ABB RobotStudio station: HandTracking_gripper_2.0.rspag

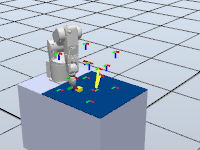
--- station ---
Station HandTrackingWithGripper (saved by RobotStudio 7.0.8743.626)
Controller Controller1, task T_ROB1: task frame (RAPID world) sits at (-300, 0, 800) mm in the station
Controller Controller1
  mechanical unit ROB_1: IRB1200_7_70_STD_02, 6 joints, base frame (0, 0, 0) mm
Layout (positions relative to the parent item):
  - IRB1200_7_70_STD_02 [mechanism, from Robots\IRB1200_7_70_STD_02.rslib] at (-300, 0, 800) mm; joint values [-0.4483, 0.9444, 0.5545, 0, 0.0719, 2.6932] (rad or m)
  - Stojalo3 [part] at (0, -390, 400) mm
  - Part_1 [part]
  - Smart_Gripper_Servo_Fingers_2_2 [mechanism] at (16, -152, 975.2) mm, rotated rx -180 ry 0 rz 0 deg; joint values [0.025] (rad or m)
      TCP Servo at (0, 0, 114.2) mm
      links: HandBase, DownFinger, UpFinger, VacuumOne, VacuumTwo
  - Part_2 [part] at (-100, 0, 0) mm
  - Part_3 [part] at (32.03, -118.48, 843.64) mm, rotated rx 0 ry 90 rz -90 deg
Attachment: Smart_Gripper_Servo_Fingers_2_2 is attached to IRB1200_7_70_STD_02 / Link6
EventTableEntry 1057: Group=, Trigger=DoFingers 1058, Actions=[EventTableActionMechanicalPose 1059], Comment=, ActivationMode=2, Cyclic=false
EventTableTriggerIO 1058: IOValue=[1], IRC5Controller=? -1, Operator=0, SignalSource=Controller1 515
EventTableActionMechanicalPose 1059: VirtualSignal=, Mechanism=Smart_Gripper_Servo_Fingers_2_2 1049, ToPoseName=Zaprto, VirtualSignalValue=[1]
EventTableEntry 1060: Group=, Trigger=DoFingers 1061, Actions=[EventTableActionMechanicalPose 1062], Comment=, ActivationMode=2, Cyclic=false
EventTableTriggerIO 1061: IOValue=[0], IRC5Controller=? -1, Operator=0, SignalSource=Controller1 515
EventTableActionMechanicalPose 1062: VirtualSignal=, Mechanism=Smart_Gripper_Servo_Fingers_2_2 1049, ToPoseName=Odprto, VirtualSignalValue=[1]
EventTableTriggerIO 1114: IOValue=[1], IRC5Controller=? -1, Operator=0, SignalSource=Controller1 515
EventTableTriggerIO 1115: IOValue=[0], IRC5Controller=? -1, Operator=0, SignalSource=Controller1 515
EventTableTriggerIO 1134: IOValue=[1], IRC5Controller=? -1, Operator=0, SignalSource=Controller1 515
EventTableTriggerIO 1135: IOValue=[0], IRC5Controller=? -1, Operator=0, SignalSource=Controller1 515
EventTableEntry 1193: Group=, Trigger=EventTableTriggerCustom 1194, Actions=[EventTableActionMove 1195], Comment=, ActivationMode=1, Cyclic=false
EventTableTriggerCustom 1194: Time=0, TriggerType=Timer
EventTableActionMove 1195: Object=Part_3 1203, GlobalTransform=[X=3.74915180455534E-33, Y=-6.12303176911189E-17, Z=-1, W=0, X=1, Y=6.12303176911189E-17, Z=0, W=0, X=6.12303176911189E-17, Y=-1, Z=6.12303176911189E-17, W=0, X=0.144379, Y=0, Z=0.86, W=1]
EventTableEntry 1196: Group=, Trigger=DoFingers 1197, Actions=[EventTableActionAttach 1198], Comment=, ActivationMode=2, Cyclic=false
EventTableTriggerIO 1197: IOValue=[1], IRC5Controller=? -1, Operator=0, SignalSource=Controller1 515
EventTableActionAttach 1198: AttachmentParent=Smart_Gripper_Servo_Fingers_2_2 1049, AttachmentChild=Part_3 1203, MountObject=false, Offset=[X=1, Y=0, Z=0, W=0, X=0, Y=1, Z=0, W=0, X=0, Y=0, Z=1, W=0, X=0, Y=0, Z=0, W=1], FlangeIndext=0, FindNearest=false
EventTableTriggerIO 1199: IOValue=[0], IRC5Controller=? -1, Operator=0, SignalSource=Controller1 515
EventTableEntry 1200: Group=, Trigger=DoFingers 1199, Actions=[EventTableActionDetach 1201], Comment=, ActivationMode=2, Cyclic=false
EventTableActionDetach 1201: AttachmentParent=Smart_Gripper_Servo_Fingers_2_2 1049, AttachmentChild=Part_3 1203
Targets, tools, work objects and paths stored in the station and not in the controller backup, written as RAPID:
! task T_ROB1
MODULE Module1
  CONST robtarget Target_30:=[[590,-205,410],[0,1,0,0],[-1,0,1,0],[9E+09,9E+09,9E+09,9E+09,9E+09,9E+09]];
  CONST robtarget Target_40:=[[590,195,410],[0,1,0,0],[0,0,-2,0],[9E+09,9E+09,9E+09,9E+09,9E+09,9E+09]];
  CONST robtarget Target_50:=[[190,195,410],[0,1,0,0],[0,0,0,0],[9E+09,9E+09,9E+09,9E+09,9E+09,9E+09]];
  CONST robtarget Target_60:=[[190,-205,10],[0,1,0,0],[0,0,0,0],[9E+09,9E+09,9E+09,9E+09,9E+09,9E+09]];
  CONST robtarget Target_70:=[[590,-205,10],[0,1,0,0],[0,0,0,0],[9E+09,9E+09,9E+09,9E+09,9E+09,9E+09]];
  CONST robtarget Target_80:=[[590,195,10],[0,1,0,0],[0,0,-2,0],[9E+09,9E+09,9E+09,9E+09,9E+09,9E+09]];
  CONST robtarget Target_90:=[[190,195,10],[0,1,0,0],[0,0,0,0],[9E+09,9E+09,9E+09,9E+09,9E+09,9E+09]];
  CONST robtarget Target_100:=[[108.00000974,170.999988771,-391.039697267],[0.000000118,0.000000013,0.70710678,0.707106782],[0,-1,2,0],[9E+09,9E+09,9E+09,9E+09,9E+09,9E+09]];
  CONST robtarget Target_110:=[[139.253700517,269.955882709,-327.170794361],[-0.000000081,0.000000036,0.707106783,0.707106779],[0,-1,-2,0],[9E+09,9E+09,9E+09,9E+09,9E+09,9E+09]];
ENDMODULE


--- Backups/Controller1/RAPID/TASK1/PROGMOD/Module1.mod ---
MODULE Module1
	PERS tooldata Servo:=[TRUE,[[0,0,114.2],[1,0,0,0]],[0.215,[8.7,12.3,49.2],[1,0,0,0],0.00021,0.00024,0.00009]];
	PERS wobjdata podlaga:=[FALSE,TRUE,"",[[590,-205,410],[0,0,-0.707106781,0.707106781]],[[0,0,0],[1,0,0,0]]];
    PERS num bReachable:=1;
    VAR num operatingmode:=1;
    VAR num waitpaint:=0;
    CONST robtarget home:=[[481.999971829,62.000001385,239.000022114],[-0.000000003,1,-0.000000021,0.000000068],[0,0,2,0],[9E+09,9E+09,9E+09,9E+09,9E+09,9E+09]];
    CONST robtarget Target_10:=[[490,-5,10],[0,0,1,0],[-1,0,-1,0],[9E+09,9E+09,9E+09,9E+09,9E+09,9E+09]];
    CONST robtarget Target_20:=[[205.90937827,223.382688175,387.01986369],[0.000000404,-0.00000012,0.707106786,0.707106776],[-1,-1,1,0],[9E+09,9E+09,9E+09,9E+09,9E+09,9E+09]];
    CONST robtarget TEsstarger:=[[181,225,-276],[0,0,0.707107,0.707107],[-1,-1,1,0],[9E+9,9E+9,9E+9,9E+9,9E+9,9E+9]];
    VAR num helpconfig:=0;
    VAR robtarget helprobottarget;
     VAR confdata cfgData;










     PROC main()
        VAR socketdev server_socket;
        VAR socketdev client_socket;
        VAR string receive_string;
        VAR string receive_string2;
        VAR string client_ip;
        VAR robtarget mytr;
        VAR string myIP:= "127.0.0.1"; !same as in config.py !!!





        SocketCreate server_socket;
        SocketBind server_socket,myIP, 55555;
        SocketListen server_socket;

        ConfL\Off;
        ConfJ\Off;
        SingArea \Wrist;

        MoveJ home,v1000,z30,Servo\WObj:=wobj0;


        ! Waiting for a connection request
         SocketAccept server_socket, client_socket\ClientAddress:=client_ip\Time:=WAIT_MAX;
         SocketSend client_socket \Str :="Robot at position "+TargetToString(home);

        WHILE TRUE DO
            !waiting to recive
            SocketReceive client_socket \Str := receive_string2;

            IF receive_string2="g" THEN
                !operating mode is in xy plane
               ! operatingmode:=0;

                IF DoFingers=0 THEN

                    SetDO DoFingers,1;
                     SocketSend client_socket \Str :="Robot grabbing";

                ELSEIF DoFingers=1 THEN
                    SetDO DoFingers,0;
                     SocketSend client_socket \Str :="Robot realising";


                ENDIF

                !TPWrite"moving set to XY plane now";


             ELSEIF receive_string2="xy" THEN
                !operating mode is in xy plane
                operatingmode:=0;
                SocketSend client_socket \Str :="operating in xy now";

                !TPWrite"moving set to XY plane now";

            ELSEIF receive_string2="xyz" THEN
                !operating mode is in xyz plane
                operatingmode:=1;
                waitpaint:=0;
                SocketSend client_socket \Str :="operating in xyz now";
                !TPWrite"moving set to XYZ now !";



            ELSE
                !MOVE

                 mytr:= StringToTargetFromxy(receive_string2); !get target from string
                 move mytr;!check if is reachable then move

            ENDIF


        ENDWHILE
        MoveJ home,v1000,z100,Servo\WObj:=wobj0;
        MoveL Target_10,v1000,z100,Servo\WObj:=wobj0;


    ERROR
        IF ERRNO=ERR_SOCK_TIMEOUT THEN
            RETRY;

        ELSEIF ERRNO=ERR_SOCK_CLOSED THEN

        SocketCreate server_socket;
        SocketBind server_socket, myIP, 55555;
        SocketListen server_socket;
            RETRY;
        ELSE
            RETRY;

        ENDIF
    UNDO
        SocketClose server_socket;
        SocketClose client_socket;
    ENDPROC


     FUNC robtarget create_robtarget(pos position)
       RETURN [position,[0,0,0.707106781,0.707106781],cfgData,[9E9,9E9,9E9,9E9,9E9,9E9]];
    ENDFUNC

    FUNC string TargetToString(robtarget target)
    VAR string tmpString;
    !pos data
    tmpString:=NumToStr (target.trans.x,0);
    AddToString tmpString,target.trans.y;
    AddToString tmpString, target.trans.z;
    ! orient data
    AddToString tmpString, target.rot.q1;
    AddToString tmpString, target.rot.q2;
    AddToString tmpString, target.rot.q3;
    AddToString tmpString, target.rot.q4;
    ! conf data
    AddToString tmpString, target.robconf.cf1;
    AddToString tmpString, target.robconf.cf4;
    AddToString tmpString, target.robconf.cf6;
    AddToString tmpString, target.robconf.cfx;
RETURN tmpString;
ENDFUNC

FUNC robtarget StringToTarget(string value)
    !CAN BE USED IF OREANTATIONS ARE NEEDED CURENTLY NOT USED
VAR robtarget tmpTarget;
VAR bool bResult;
VAR num posX;
VAR num posY;
VAR num posZ;
VAR num posQ1;
VAR num posQ2;
VAR num posQ3;
VAR num posQ4;
VAR num poscf1;
VAR num poscf4;
VAR num poscf6;
VAR num poscfx;
! Find split positions in string

posX:=StrFind (value, 1,";");
posY:=StrFind (value, posX+1,";");
posZ:=StrFind (value, posY+1,";");
posQ1:=StrFind (value, posZ+1,";");
posQ2:=StrFind(value, posQ1+1,";");
posQ3:=StrFind (value,posQ2+1,";");
posQ4:=Strfind(value, posQ3+1,";");
poscf1:=StrFind(value, posQ4+1,";");
poscf4:=StrFind(value, poscf1+1,";");
poscf6:=StrFind(value, poscf4+1,";");
poscfx:=StrFind(value,poscf6+1, ";");
! read all strings
! pos data
bResult:=StrToval(StrPart(value,1,posX-1), tmpTarget.trans.x);
bResult:=StrToVal(StrPart(value,posX+1, posY-posX-1), tmpTarget.trans.y);
bResult:=StrToVal(StrPart(value,posY+1, posZ-posY -1), tmpTarget.trans.z);
! orient data
bResult:=StrToVal(StrPart(value, posZ+1, posQ1-posz-1), tmpTarget.rot.q1);
bResult:=StrToval (StrPart(value,posQ1+1, posQ2-posQ1-1), tmpTarget.rot.q2);
bResult:=StrToVal(StrPart(value,posQ2+1, posQ3-posQ2-1), tmpTarget.rot.q3);
bResult:=StrToVal(StrPart(value,posQ3+1,posQ4-posQ3-1), tmpTarget.rot.q4);
! conf data
bResult:=StrToVal(StrPart(value,posQ4+1, poscf1-posQ4-1), tmpTarget.robconf.cf1);
bResult:=StrToVal(StrPart(value, poscf1+1,poscf4-poscf1-1), tmpTarget.robconf.cf4);
bResult:=StrToval(StrPart(value,poscf4+1,poscf6-poscf4-1), tmpTarget.robconf.cf6);
bResult:=StrToVal(StrPart(value,poscf6+1,poscfx-poscf6-1), tmpTarget.robconf.cfx);
RETURN tmpTarget;

ERROR
    !RETURN !Target_20;



ENDFUNC

FUNC robtarget StringToTargetFromxy(string value)
VAR pos tmpPos;
VAR robtarget tmpTarget;
VAR bool bResult;
VAR num posX;
VAR num posY;
VAR num posZ;
VAR num xxx;
VAR num yyy;
VAR num zzz:=-330;
! Find split positions in string

posX:=StrFind (value, 1,";");
posY:=StrFind (value, posX+1,";");
IF operatingmode=1 THEN
posZ:=StrFind (value, posY+1,";");
ENDIF

! pos data
bResult:=StrToval(StrPart(value,1,posX-1), tmpPos.x);

tmpPos.x:=tmpPos.x;

bResult:=StrToVal(StrPart(value,posX+1, posY-posX-1), tmpPos.y);

tmpPos.y:=tmpPos.y;

IF operatingmode=1 THEN
bResult:=StrToVal(StrPart(value,posY+1, posZ-posY -1), tmpPos.z);

tmpPos.z:=-tmpPos.z;

ELSE
tmpPos.z:=zzz; !z is set to 0
ENDIF
tmpTarget:=create_robtarget(tmpPos);
RETURN tmpTarget;

ERROR
   ! RETURN Target_20;!middle target of error
ENDFUNC

PROC AddToString(INOUT string inString,num value)
inString:=inString+";"+NumToStr(value,0);
ENDPROC

PROC move(robtarget target)
     VAR bool aotoconfiggg;
     VAR bool precheck:=FALSE;
     precheck:=simplecheck(target,Servo);

     !IF precheck=FALSE THEN
    !aotoconfiggg:= calcconfiguration(target,Servo);
     !IF aotoconfiggg=TRUE THEN
      !   target.robconf:=cfgData;

    !CheckReachable target,Servo;
     !      IF bReachable=2 THEN
                !notreachable
      !          TPWrite"not reachable";
       !    ELSEIF bReachable=1 THEN
                !reachable start moving
        !        MoveJ target,v2000,z10,Servo\WObj:=podlaga;

                !move target;
         ! ENDIF
          ! ELSE
        ! RETURN;
     !ENDIF

     !ELSE
          MoveJ target,v2000,z10,Servo\WObj:=podlaga;

     !ENDIF

    ERROR
        TPWrite"error in move";
        TRYNEXT;

ENDPROC


 PROC CheckReachable(robtarget myRobtarget,PERS tooldata ToolReach1,\PERS wobjdata WobjReach1)

      VAR jointtarget jntReach1;



      bReachable:=1;

            jntReach1:=CalcJointT(myRobtarget,ToolReach1);

      RETURN;
      ERROR


         IF ERRNO=ERR_OUTSIDE_REACH THEN

                bReachable:=2;
               TRYNEXT;

        ENDIF
         IF ERRNO=ERR_ROBLIMIT THEN

                bReachable:=2;
               TRYNEXT;

        ENDIF
        bReachable:=2;
        RETURN;
  ENDPROC

  FUNC bool calcconfiguration(robtarget rtg,PERS tooldata ToolReach2,\PERS wobjdata WobjReach2)

      VAR bool bFound:=FALSE;
      VAR bool passed:=FALSE;
      VAR bool loop:=TRUE;

    WHILE   loop DO
    FOR  c1 FROM -2 TO 1 STEP 1 DO
        FOR c2 FROM -3 TO 2 STEP 1 DO
            FOR c3 FROM -5 TO 4 STEP 1 DO
                rtg.robconf := [c1, c2, c3, 0];
                passed:=simplecheck(rtg,ToolReach2);

                IF(passed=TRUE) THEN
                    bFound := TRUE;
                    cfgData := [c1, c2, c3, 0];
                    TPWrite ValToStr(cfgData);
                    loop:=FALSE;


                ENDIF
                IF rtg.robconf=[1, 2, 4, 0] THEN
                    loop:=FALSE;

                ENDIF
            ENDFOR
        ENDFOR
    ENDFOR
    ENDWHILE

    IF bfound THEN
        RETURN TRUE;

    ELSE
        RETURN FALSE;

    ENDIF
  ENDFUNC

  FUNC bool simplecheck(robtarget rtgg,PERS tooldata ToolReach1,\PERS wobjdata WobjReach1)
      VAR jointtarget jntReach2;
            jntReach2:=CalcJointT(rtgg,ToolReach1);


      RETURN TRUE;
    ERROR
    RETURN FALSE;

  ENDFUNC


ENDMODULE

--- Backups/Controller1/SYSPAR/EIO.cfg ---
EIO:CFG_1.0:6:1::
#
EIO_SIGNAL:

      -Name "DoFingers" -SignalType "DO" -Access "All"
